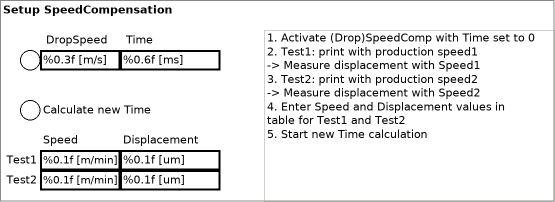
VISUALIZATION _VISU_DropSpeedComp_Setup  // 555x202
VAR_IN_OUT
	mInst : FB_DropSpeedComp;
END_VAR
    Rectangle (0,0 555x202)
    Ellipse (20,50 20x20), tooltip "Enable Correction"
        toggle mInst.bEnable p2164770859=TRUE
    Rectangle (40,50 80x20), "%0.3f [m/s]", tooltip "DropSpeed", text variable: mInst.fDropSpeed
        OnMouseClick: write the text variable via Default
    Rectangle (120,50 100x20), "%0.6f [ms]", tooltip "Dead/Add Time", text variable: mInst.fDropSpeedDeadTime
        OnMouseClick: write the text variable via Default
    Rectangle (123,30 78x20), "Time"
    Rectangle (43,30 78x20), "DropSpeed"
    Ellipse (20,100 20x20), tooltip "Calculate new time"
        tap mInst.bCalcDeadTime
    Rectangle (40,150 80x20), "%0.1f [m/min]", text variable: mInst.fTestSpeed[1]
        OnMouseClick: write the text variable via Default
    Rectangle (40,170 80x20), "%0.1f [m/min]", text variable: mInst.fTestSpeed[2]
        OnMouseClick: write the text variable via Default
    Rectangle (40,130 78x20), "Speed"
    Rectangle (120,150 100x20), "%0.1f [um]", text variable: mInst.fTestDisplacement[1]
        OnMouseClick: write the text variable via Default
    Rectangle (120,170 100x20), "%0.1f [um]", text variable: mInst.fTestDisplacement[2]
        OnMouseClick: write the text variable via Default
    Rectangle (120,130 100x20), "Displacement"
    Rectangle (0,0 256x20), "Setup SpeedCompensation"
    Rectangle (40,100 150x20), "Calculate new Time"
    Rectangle (0,150 40x20), "Test1"
    Rectangle (0,170 40x20), "Test2"
    Textfield (264,30 291x172), "1. Activate (Drop)SpeedComp with Time set to 0 2. Test1: print with production speed1 -> Measure displacement with Speed1 3. Test2: print with production speed2 -> Measure displacement with Speed2 4. Enter Speed and Displacement values in table for Test1 and Test2 5. Start new Time calculation"
END_VISUALIZATION

(* stored: Version 1.1.0.1, ProductVersion 3.1.4024.11
   Visu _VISU_DropSpeedComp_Setup: Id {c469460c-51b8-454b-8e1b-2c03811413e2} *)
